FUNCTION_BLOCK TN_SC_WRITE_EOS
VAR
	TN_SC_WRITE : TN_SC_WRITE;
END_VAR
VAR_INPUT
	Iby_ATTR : BYTE;
	Ist_STRING : STRING;
END_VAR
VAR_IN_OUT
	Xus_TN_SCREEN : us_TN_SCREEN;
END_VAR

(*
version 1.0		10. mai 2010
programmer		ks
tested by		ks

TN_SC_WRITE_EOS schreibt einem Text an das Ende des zuletzt geschreibene Texts 
*)

TN_SC_WRITE(Iin_Y := Xus_TN_SCREEN.in_EOS_Offset / 80, (* aktuelle Zeile ausrechnen *)
			Iin_X := Xus_TN_SCREEN.in_EOS_Offset MOD 80, (* aktuelle Spalte ausrechnen *)
			Iby_ATTR := Iby_ATTR,
			Ist_STRING := Ist_STRING,
			Xus_TN_SCREEN := Xus_TN_SCREEN);

(* revision history
ks	10. mai. 2010	rev 1.0
	original version
*)

END_FUNCTION_BLOCK

(* stored: Version 1.1.0.1, ProductVersion 3.1.4024.0
   POU TN_SC_WRITE_EOS: Id {78a96012-804d-41ae-8a63-c8ec78d31d52}, SpecialFunc None *)
